PROGRAM MAIN
VAR
	diKapSensor1 AT %I* : BOOL ;
	diKapSensor2 AT %I* : BOOL ;

	bMinneKapSensor1 : BOOL := 0 ;
	bMinneKapSensor2 : BOOL := 0 ;
	
END_VAR

bMinneKapSensor1 := diKapSensor1 ;
bMinneKapSensor2 := diKapSensor2 ;

bMinneKapSensor1 := diKapSensor1 AND diKapSensor2 ;
bMinneKapSensor2 := diKapSensor1 OR diKapSensor2 ;

END_PROGRAM

(* stored: Version 1.1.0.1, ProductVersion 3.1.4024.9
   POU MAIN: Id {0ad9fa93-8e95-4f2c-9f05-28f2199517bd}, SpecialFunc None *)
